PROGRAM MAIN
VAR
	tpImAPLC : TP := (PT:=T#10S);
	//stDiag	:	ST_fbDiagnostics;
	
	//FEEM1PitchControl	:	FB_PitchControl;
	FEEM1PitchControl	:	FB_PitchControl;
	FEEM1Y_GantryControl	:	FB_Gantry;
	FEEM1X_GantryControl	:	FB_Gantry;
	FEEM2PitchControl	    :	FB_PitchControl;
	FEEM2Y_GantryControl	:	FB_Gantry;
	FEEM2X_GantryControl	:	FB_Gantry;
	
	FEEM1_BenderControl		:	FB_PTP;
	
	// Expert mode permits direct access to individual acutators.
	ExpertMode	:	BOOL := FALSE;
	DirectPiezoMode: BOOL := FALSE;
	
	//Limit switch evaluation blocks
	fbM1Y1LS	:	FB_LimitSwitchState;
	fbM1Y2LS	:	FB_LimitSwitchState;
	fbM1X1LS	:	FB_LimitSwitchState;
	fbM1X2LS	:	FB_LimitSwitchState;
	fbM1P1LS	:	FB_LimitSwitchState;
	
	fbM2Y1LS	:	FB_LimitSwitchState;
	fbM2Y2LS	:	FB_LimitSwitchState;
	fbM2X1LS	:	FB_LimitSwitchState;
	fbM2X2LS	:	FB_LimitSwitchState;
	fbM2P1LS	:	FB_LimitSwitchState;	
	
	//Drive CoE Fb
	fbY1CoE	:	FB_ElmoGDCBellCoE;
	fbY2CoE	:	FB_ElmoGDCBellCoE;
	
	fbX1CoE	:	FB_ElmoGDCBellCoE;
	fbX2CoE	:	FB_ElmoGDCBellCoE;
	
	fbP1CoE	:	FB_ElmoGDCBellCoE;
	fbB1CoE	:	FB_ElmoGDCBellCoE;
	
	
	//Init params trigger
	rtInitParams	:	R_TRIG;
	
	//Test Parameters
		rStepSize: REAL;
	SettleTime: TON := (
	PT:=T#2s);
	TestUpperVoltage: REAL := 100;
	TestLowerVoltage: REAL := 10;
	xRunPiezoRepeatTest: BOOL;
	
	//Drive reference initializations
	fbInitDriveRef	:	FB_InitDriveRefs;
	
END_VAR

//System IO
/////////////////////////////
p_ModbusRx_OutputCoils();
p_ModbusRx_PLCMemory();

//DriveCoEIO(); //This is now done in the FB_PTP block
//InitParams
////////////////////
rtInitParams(CLK:=gFirstPass);
IF rtInitParams.Q THEN
	Init_FEEM1();
	Init_FEEM2();
	gFirstPass := FALSE;
END_IF

//System Error Handling
/////////////////////////////////////
//SystemErrorSummary(); //Check this action for a summary of all system faults
					  
//SystemError();

//Driver Parameter Verification
/////////////////////////////////////

//Gantry Interlock Logic
/////////////////////////////////////
	//SimGantry.VAxis.i_xMotorInterlock := TRUE;
	//SimGantry.PAxis.i_xMotorInterlock := TRUE;
	//SimGantry.SAxis.i_xMotorInterlock := TRUE;
	//P_GantryDiffSup(); //This is now done in FB_Gantry block
LimitSwitchIO();
	
// Pitch control
/////////////////////////////////////
FEEM1PitchControl(Pitch:=HOMS1_Pitch, DirectPiezoMode:=(ExpertMode AND DirectPiezoMode));
FEEM2PitchControl(Pitch:=HOMS2_Pitch, DirectPiezoMode:=(ExpertMode AND DirectPiezoMode));

// Bender control
//////////////////////////////////
FEEM1_BenderControl(Stepper:=HOMS1_Bender);


//Y motion
/////////////////////////////////////
FEEM1Y_GantryControl(Gantry:=HOMS1_YGantry);
FEEM2Y_GantryControl(Gantry:=HOMS2_YGantry);
	
//X Motion
/////////////////////////////////////
FEEM1X_GantryControl(Gantry:=HOMS1_XGantry);
FEEM2X_GantryControl(Gantry:=HOMS2_XGantry);

//EPICS Tx Update
////////////////////
p_ModbusTx_InputCoils();
//p_ModbusTx_OutputCoils();
p_ModbusTx_InputReg();
p_ModbusTx_PLCMemory();

ACTION Init_FEEM1:
//FEE-M1
///////////////////////////

//Initialize Center positions
HOMS1_XGantry.PAxis.cCenter := HOMS1_XGantry_PAxisCenter;
HOMS1_XGantry.SAxis.cCenter := HOMS1_XGantry_SAxisCenter;
HOMS1_YGantry.PAxis.cCenter := HOMS1_YGantry_PAxisCenter;
HOMS1_YGantry.SAxis.cCenter := HOMS1_YGantry_SAxisCenter;

//Initialize ELMO Drive references
fbInitDriveRef(stCoE:=HOMS1_XGantry.PAxis.stCoE);
fbInitDriveRef(stCoE:=HOMS1_XGantry.SAxis.stCoE);
fbInitDriveRef(stCoE:=HOMS1_YGantry.PAxis.stCoE);
fbInitDriveRef(stCoE:=HOMS1_YGantry.SAxis.stCoE);
fbInitDriveRef(stCoE:=HOMS1_Pitch.Stepper.stCoE);

//Initialze Drive Speeds and Accelerations
//////////////////////////////////////////
HOMS1_XGantry.PAxis.fAcceleration := 0.02;
HOMS1_XGantry.SAxis.fAcceleration := 0.02;
HOMS1_YGantry.PAxis.fAcceleration := 0.02;
HOMS1_YGantry.SAxis.fAcceleration := 0.02;

HOMS1_XGantry.PAxis.fDeceleration := 0.02;
HOMS1_XGantry.SAxis.fDeceleration := 0.02;
HOMS1_YGantry.PAxis.fDeceleration := 0.02;
HOMS1_YGantry.SAxis.fDeceleration := 0.02;

HOMS1_XGantry.PAxis.fVelocity := 0.1;
HOMS1_XGantry.SAxis.fVelocity := 0.1;
HOMS1_YGantry.PAxis.fVelocity := 0.1;
HOMS1_YGantry.SAxis.fVelocity := 0.1;

HOMS1_Pitch.Stepper.fAcceleration := 0.02;
HOMS1_Pitch.Stepper.fDeceleration := 0.02;
HOMS1_Pitch.Stepper.fVelocity     := 0.02;


//Initialize Piezo Driver
/////////////////////////////////////
HOMS1_Pitch.Piezo.stPIParams.fKp := 1;
HOMS1_Pitch.Piezo.stPIParams.tTn := T#100mS;
HOMS1_Pitch.Piezo.stPIParams.fOutMaxLimit := 1;
HOMS1_Pitch.Piezo.stPIParams.fOutMinLimit := -1;
END_ACTION

ACTION Init_FEEM2:
//FEE-M2
///////////////////////////

//Initialize Center positions
HOMS2_XGantry.PAxis.cCenter := HOMS2_XGantry_PAxisCenter;
HOMS2_XGantry.SAxis.cCenter := HOMS2_XGantry_SAxisCenter;
HOMS2_YGantry.PAxis.cCenter := HOMS2_YGantry_PAxisCenter;
HOMS2_YGantry.SAxis.cCenter := HOMS2_YGantry_SAxisCenter;

//Initialize ELMO Drive references
fbInitDriveRef(stCoE:=HOMS2_XGantry.PAxis.stCoE);
fbInitDriveRef(stCoE:=HOMS2_XGantry.SAxis.stCoE);
fbInitDriveRef(stCoE:=HOMS2_YGantry.PAxis.stCoE);
fbInitDriveRef(stCoE:=HOMS2_YGantry.SAxis.stCoE);
fbInitDriveRef(stCoE:=HOMS2_Pitch.Stepper.stCoE);

//Initialze Drive Speeds and Accelerations
//////////////////////////////////////////
HOMS2_XGantry.PAxis.fAcceleration := 0.02;
HOMS2_XGantry.SAxis.fAcceleration := 0.02;
HOMS2_YGantry.PAxis.fAcceleration := 0.02;
HOMS2_YGantry.SAxis.fAcceleration := 0.02;

HOMS2_XGantry.PAxis.fDeceleration := 0.02;
HOMS2_XGantry.SAxis.fDeceleration := 0.02;
HOMS2_YGantry.PAxis.fDeceleration := 0.02;
HOMS2_YGantry.SAxis.fDeceleration := 0.02;

HOMS2_XGantry.PAxis.fVelocity := 0.1;
HOMS2_XGantry.SAxis.fVelocity := 0.1;
HOMS2_YGantry.PAxis.fVelocity := 0.1;
HOMS2_YGantry.SAxis.fVelocity := 0.1;

HOMS2_Pitch.Stepper.fAcceleration := 0.02;
HOMS2_Pitch.Stepper.fDeceleration := 0.02;
HOMS2_Pitch.Stepper.fVelocity     := 0.02;

//Initialize Piezo Driver
/////////////////////////////////////
HOMS2_Pitch.Piezo.stPIParams.fKp := 1;
HOMS2_Pitch.Piezo.stPIParams.tTn := T#100mS;
HOMS2_Pitch.Piezo.stPIParams.fOutMaxLimit := 1;
HOMS2_Pitch.Piezo.stPIParams.fOutMinLimit := -1;
END_ACTION

ACTION LimitSwitchIO:
//FEE M1
///////////////////
fbM1Y1LS(diInputs:=HOMS1_YGantry.PAxis.diInputs, 
xHiLS=>HOMS1_YGantry.PAxis.xHiLS,
xLoLS=>HOMS1_YGantry.PAxis.xLoLS);

fbM1Y2LS(diInputs:=HOMS1_YGantry.SAxis.diInputs, 
xHiLS=>HOMS1_YGantry.SAxis.xHiLS,
xLoLS=>HOMS1_YGantry.SAxis.xLoLS);

fbM1X1LS(diInputs:=HOMS1_XGantry.PAxis.diInputs, 
xHiLS=>HOMS1_XGantry.PAxis.xHiLS,
xLoLS=>HOMS1_XGantry.PAxis.xLoLS);

fbM1X2LS(diInputs:=HOMS1_XGantry.SAxis.diInputs, 
xHiLS=>HOMS1_XGantry.SAxis.xHiLS,
xLoLS=>HOMS1_XGantry.SAxis.xLoLS);

fbM1P1LS(diInputs:=HOMS1_Pitch.stepper.diInputs,
xHiLS=>HOMS1_Pitch.Stepper.xHiLS,
xLoLS=>HOMS1_Pitch.Stepper.xLoLS);


//FEE M2
//////////////////////////
fbM2Y1LS(diInputs:=HOMS2_YGantry.PAxis.diInputs, 
xHiLS=>HOMS2_YGantry.PAxis.xHiLS,
xLoLS=>HOMS2_YGantry.PAxis.xLoLS);

fbM2Y2LS(diInputs:=HOMS2_YGantry.SAxis.diInputs, 
xHiLS=>HOMS2_YGantry.SAxis.xHiLS,
xLoLS=>HOMS2_YGantry.SAxis.xLoLS);

fbM2X1LS(diInputs:=HOMS2_XGantry.PAxis.diInputs, 
xHiLS=>HOMS2_XGantry.PAxis.xHiLS,
xLoLS=>HOMS2_XGantry.PAxis.xLoLS);

fbM2X2LS(diInputs:=HOMS2_XGantry.SAxis.diInputs, 
xHiLS=>HOMS2_XGantry.SAxis.xHiLS,
xLoLS=>HOMS2_XGantry.SAxis.xLoLS);

fbM2P1LS(diInputs:=HOMS2_Pitch.stepper.diInputs,
xHiLS=>HOMS2_Pitch.Stepper.xHiLS,
xLoLS=>HOMS2_Pitch.Stepper.xLoLS);
END_ACTION

END_PROGRAM

(* stored: Version 1.1.0.1, ProductVersion 3.1.4020.12
   POU MAIN: Id {ea0bf136-bb68-48b6-99e0-4530d55408e2}, SpecialFunc None
   Action Init_FEEM1: Id {a11eaaff-25fb-4e40-9807-fb1f683338da}
   Action Init_FEEM2: Id {5f4f0886-bfe6-466e-ab0f-beab0308d09d}
   Action LimitSwitchIO: Id {f9e468fa-ee02-4f8a-956e-139b70621257} *)
